// TIA Portal V17 export
// export: Created 2025-03-07T09:18:52.3547391Z, ExportSetting WithDefaults, DisplayName Totally Integrated Automation Portal, DisplayVersion V17 Update 8, DisplayName TIA Portal Openness, DisplayVersion V17 Update 8, DisplayName TIA Portal Version Control Interface, DisplayVersion V17, DisplayName SINAMICS Startdrive Advanced, DisplayVersion V17 SP2, DisplayName SINAMICS Startdrive G110M, G120, G120C, G120D, G120P, G115D, DisplayVersion V17 SP2, DisplayName SINAMICS Startdrive G130, G150, S120, S150, SINAMICS MV, S210, DisplayVersion V17 SP2, DisplayName STEP 7 Professional, DisplayVersion V17 Update 8, DisplayName SINUMERIK ONE STEP 7 Toolbox, DisplayVersion V17 Update 12, DisplayName SINUMERIK 840D sl STEP 7 Toolbox, DisplayVersion V17 Update 12, DisplayName STEP 7 Safety, DisplayVersion V17 Update 6, DisplayName WinCC Advanced, DisplayVersion V17 Update 8
FUNCTION "FC20000_LASER_SYSTEM" : Void   // FC20000, LAD
{ S7_Optimized_Access := 'TRUE' }
VERSION : 0.1
// stored: AutoNumber false, IsIECCheckEnabled false, SetENOAutomatically false, UDAEnableTagReadback false
BEGIN

REGION Network 1: CALL FC20200_LASER_TRUMPF_READY
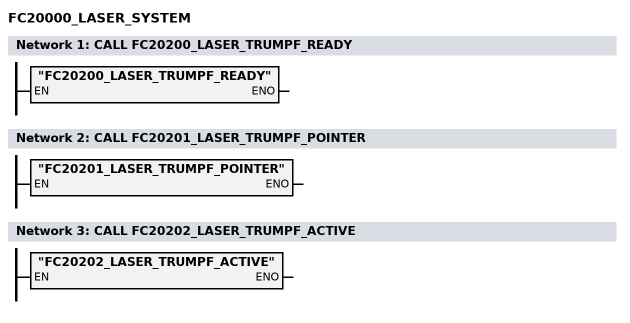
   RUNG wire#powerrail
      "FC20200_LASER_TRUMPF_READY"()
   END_RUNG
   // the same network as SCL:
   "FC20200_LASER_TRUMPF_READY"();
END_REGION

REGION Network 2: CALL FC20201_LASER_TRUMPF_POINTER
   RUNG wire#powerrail
      "FC20201_LASER_TRUMPF_POINTER"()
   END_RUNG
   // the same network as SCL:
   "FC20201_LASER_TRUMPF_POINTER"();
END_REGION

REGION Network 3: CALL FC20202_LASER_TRUMPF_ACTIVE
   RUNG wire#powerrail
      "FC20202_LASER_TRUMPF_ACTIVE"()
   END_RUNG
   // the same network as SCL:
   "FC20202_LASER_TRUMPF_ACTIVE"();
END_REGION
END_FUNCTION
